// TIA Portal project "PID_TankLevel" (V16)

(* hardware
DEVICE "S71500/ET200MP-Station_1"  S7-1500 station
   slot 0: "Profilschiene_0"  6ES7 590-1***0-0AA0
   slot 1: "PLC_1"  CPU 1511-1 PN  6ES7 511-1AK00-0AB0  V1.8
   slot 2: "AI 8xU/I/RTD/TC ST_1"  AI 8xU/I/RTD/TC ST  6ES7 531-7KF00-0AB0  V2.0
   slot 3: "AI 8xU/I/RTD/TC ST_2"  AI 8xU/I/RTD/TC ST  6ES7 531-7KF00-0AB0  V2.0
   slot 4: "AI 8xU/I/RTD/TC ST_3"  AI 8xU/I/RTD/TC ST  6ES7 531-7KF00-0AB0  V2.0
   slot 5: "AI 8xU/I/RTD/TC ST_4"  AI 8xU/I/RTD/TC ST  6ES7 531-7KF00-0AB0  V2.0
   slot 6: "DI 16x24VDC BA_1"  DI 16x24VDC BA  6ES7 521-1BH10-0AA0  V1.0
*)

// ===== PLC "PLC_1"  CPU 1511-1 PN =====

VAR_GLOBAL   // PLC tag table "Standard-Variablentabelle"
   "System_Byte" AT %MB1 : Byte;
   "FirstScan" AT %M1.0 : Bool;
   "DiagStatusUpdate" AT %M1.1 : Bool;
   "AlwaysTRUE" AT %M1.2 : Bool;
   "AlwaysFALSE" AT %M1.3 : Bool;
   "Clock_Byte" AT %MB0 : Byte;
   "Clock_10Hz" AT %M0.0 : Bool;
   "Clock_5Hz" AT %M0.1 : Bool;
   "Clock_2.5Hz" AT %M0.2 : Bool;
   "Clock_2Hz" AT %M0.3 : Bool;
   "Clock_1.25Hz" AT %M0.4 : Bool;
   "Clock_1Hz" AT %M0.5 : Bool;
   "Clock_0.625Hz" AT %M0.6 : Bool;
   "Clock_0.5Hz" AT %M0.7 : Bool;
END_VAR

VAR_GLOBAL   // PLC tag table "INPUTS"
   "StartButton" AT %I0.0 : Bool;
   "ResetButton" AT %I0.1 : Bool;
   "StopButton" AT %I0.2 : Bool;
   "FactoryIORunning" AT %I0.3 : Bool;
   "LevelMeter" AT %ID30 : Real;
   "FlowMeter" AT %ID34 : Real;
   "SetPoint" AT %ID38 : Real;
END_VAR

VAR_GLOBAL   // PLC tag table "OUTPUTS"
   "StartLight" AT %Q0.0 : Bool;
   "ResetLight" AT %Q0.1 : Bool;
   "StopLight" AT %Q0.2 : Bool;
   "FillValve" AT %QD30 : Real;
   "DischargeValve" AT %QD34 : Real;
   "SP" AT %QD38 : DInt;
   "PV" AT %QD42 : DInt;
END_VAR

VAR_GLOBAL   // PLC tag table "SystemTags"
   "LevelMeter_Scaled" AT %MD30 : DInt;
   "FlowMeter_Scaled" AT %MD34 : DInt;
   "SetPoint_Scaled" AT %MD38 : DInt;
   "FillValve_Scaled" AT %MD42 : DInt;
   "DischargeValve_Scaled" AT %MD46 : DInt;
END_VAR

VAR_GLOBAL   // PLC tag table "GeneralTags"
   "System ON/OFF" AT %M100.0 : Bool;
END_VAR

ORGANIZATION_BLOCK "Main"   // OB1, LAD, ProgramCycle
TITLE = "Main Program Sweep (Cycle)"
{ S7_Optimized_Access := 'TRUE' }
VERSION : 0.1
   VAR_INPUT
      Initial_Call : Bool;   // Initial call of this OB
      Remanence : Bool;   // =True, if remanent data are available
   END_VAR
BEGIN

REGION Network 2
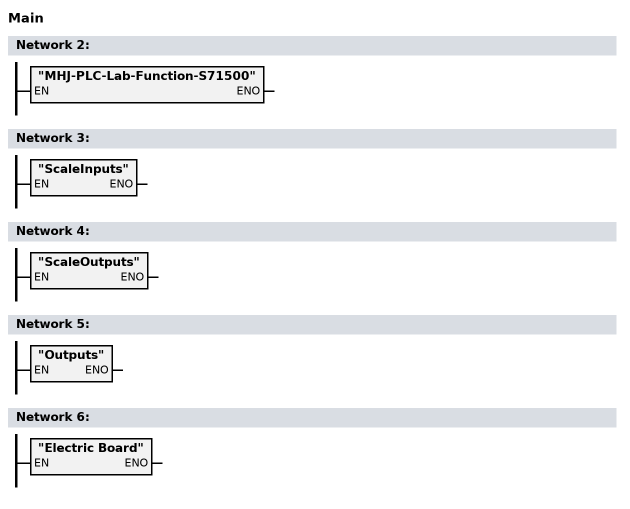
   RUNG wire#powerrail
      "MHJ-PLC-Lab-Function-S71500"()
   END_RUNG
   // the same network as SCL:
   "MHJ-PLC-Lab-Function-S71500"();
END_REGION

REGION Network 3
   RUNG wire#powerrail
      "ScaleInputs"()
   END_RUNG
   // the same network as SCL:
   "ScaleInputs"();
END_REGION

REGION Network 4
   RUNG wire#powerrail
      "ScaleOutputs"()
   END_RUNG
   // the same network as SCL:
   "ScaleOutputs"();
END_REGION

REGION Network 5
   RUNG wire#powerrail
      "Outputs"()
   END_RUNG
   // the same network as SCL:
   "Outputs"();
END_REGION

REGION Network 6
   RUNG wire#powerrail
      "Electric Board"()
   END_RUNG
   // the same network as SCL:
   "Electric Board"();
END_REGION
END_ORGANIZATION_BLOCK

// folder: INPUTS&OUTPUTS

FUNCTION "ScaleInputs" : Void   // FC1, LAD
{ S7_Optimized_Access := 'TRUE' }
VERSION : 0.1
   VAR_TEMP
      temp_levelmeter : Real;
      temp_setpoint : Real;
   END_VAR
BEGIN

REGION Network 2
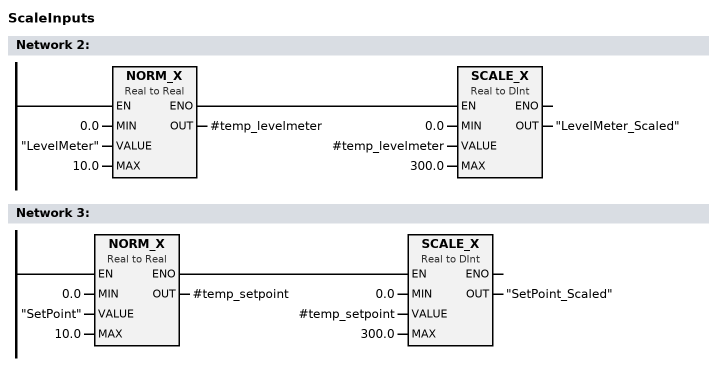
   RUNG wire#powerrail
      { S7_Templates := "[SrcType := Real, DestType := Real]" } Normalize(min := 0.0, value := "LevelMeter", max := 10.0, out => #temp_levelmeter)
      { S7_Templates := "[SrcType := Real, DestType := DInt]" } Scale(min := 0.0, value := #temp_levelmeter, max := 300.0, out => "LevelMeter_Scaled")
   END_RUNG
   // the same network as SCL:
   #temp_levelmeter := NORM_X(MIN := 0.0, VALUE := "LevelMeter", MAX := 10.0);
   "LevelMeter_Scaled" := SCALE_X(MIN := 0.0, VALUE := #temp_levelmeter, MAX := 300.0);
END_REGION

REGION Network 3
   RUNG wire#powerrail
      { S7_Templates := "[SrcType := Real, DestType := Real]" } Normalize(min := 0.0, value := "SetPoint", max := 10.0, out => #temp_setpoint)
      { S7_Templates := "[SrcType := Real, DestType := DInt]" } Scale(min := 0.0, value := #temp_setpoint, max := 300.0, out => "SetPoint_Scaled")
   END_RUNG
   // the same network as SCL:
   #temp_setpoint := NORM_X(MIN := 0.0, VALUE := "SetPoint", MAX := 10.0);
   "SetPoint_Scaled" := SCALE_X(MIN := 0.0, VALUE := #temp_setpoint, MAX := 300.0);
END_REGION
END_FUNCTION

FUNCTION "Outputs" : Void   // FC2, LAD
{ S7_Optimized_Access := 'TRUE' }
VERSION : 0.1
BEGIN

REGION Network 2
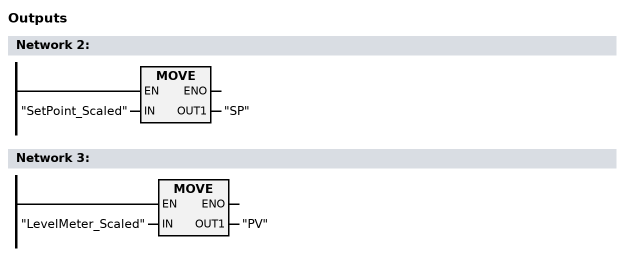
   RUNG wire#powerrail
      Move(in := "SetPoint_Scaled", out1 => "SP")
   END_RUNG
   // the same network as SCL:
   "SP" := "SetPoint_Scaled";
END_REGION

REGION Network 3
   RUNG wire#powerrail
      Move(in := "LevelMeter_Scaled", out1 => "PV")
   END_RUNG
   // the same network as SCL:
   "PV" := "LevelMeter_Scaled";
END_REGION
END_FUNCTION

FUNCTION "ScaleOutputs" : Void   // FC3, LAD
{ S7_Optimized_Access := 'TRUE' }
VERSION : 0.1
   VAR_TEMP
      temp_fillvalve : Real;
      temp_dischargevalve : Real;
   END_VAR
BEGIN

REGION Network 2
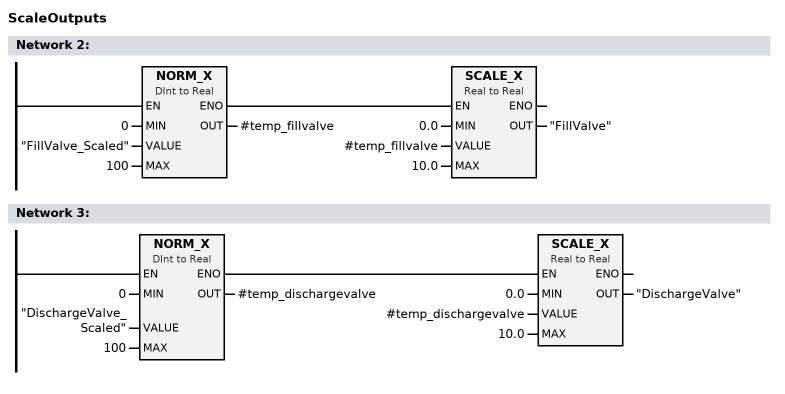
   RUNG wire#powerrail
      { S7_Templates := "[SrcType := DInt, DestType := Real]" } Normalize(min := 0, value := "FillValve_Scaled", max := 100, out => #temp_fillvalve)
      { S7_Templates := "[SrcType := Real, DestType := Real]" } Scale(min := 0.0, value := #temp_fillvalve, max := 10.0, out => "FillValve")
   END_RUNG
   // the same network as SCL:
   #temp_fillvalve := NORM_X(MIN := 0, VALUE := "FillValve_Scaled", MAX := 100);
   "FillValve" := SCALE_X(MIN := 0.0, VALUE := #temp_fillvalve, MAX := 10.0);
END_REGION

REGION Network 3
   RUNG wire#powerrail
      { S7_Templates := "[SrcType := DInt, DestType := Real]" } Normalize(min := 0, value := "DischargeValve_Scaled", max := 100, out => #temp_dischargevalve)
      { S7_Templates := "[SrcType := Real, DestType := Real]" } Scale(min := 0.0, value := #temp_dischargevalve, max := 10.0, out => "DischargeValve")
   END_RUNG
   // the same network as SCL:
   #temp_dischargevalve := NORM_X(MIN := 0, VALUE := "DischargeValve_Scaled", MAX := 100);
   "DischargeValve" := SCALE_X(MIN := 0.0, VALUE := #temp_dischargevalve, MAX := 10.0);
END_REGION
END_FUNCTION

// folder: SYSTEM BLOCKS

FUNCTION "Electric Board" : Void   // FC4, LAD
{ S7_Optimized_Access := 'TRUE' }
VERSION : 0.1
BEGIN

REGION Network 2
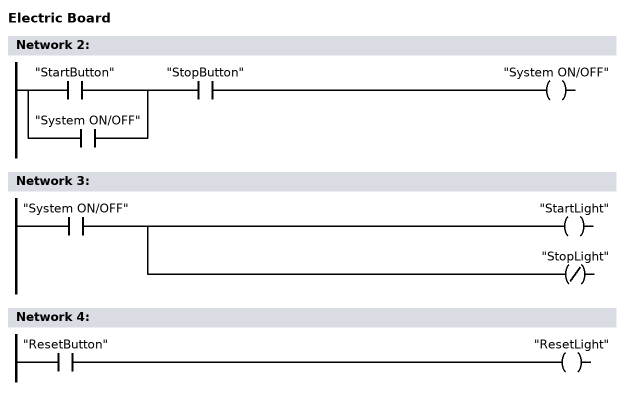
   RUNG wire#powerrail
      Contact( "StartButton" )
      wire#w1
      Contact( "StopButton" )
      Coil( "System ON/OFF" )
   END_RUNG
   RUNG wire#powerrail
      Contact( "System ON/OFF" )
   END_RUNG wire#w1
   // the same network as SCL:
   "System ON/OFF" := ("StartButton" OR "System ON/OFF") AND "StopButton";
END_REGION

REGION Network 3
   RUNG wire#powerrail
      Contact( "System ON/OFF" )
      wire#w1
      Coil( "StartLight" )
   END_RUNG
   RUNG wire#w1
      I_Coil( "StopLight" )
   END_RUNG
   // the same network as SCL:
   "StartLight" := "System ON/OFF";
   "StopLight" := NOT "System ON/OFF";
END_REGION

REGION Network 4
   RUNG wire#powerrail
      Contact( "ResetButton" )
      Coil( "ResetLight" )
   END_RUNG
   // the same network as SCL:
   "ResetLight" := "ResetButton";
END_REGION
END_FUNCTION

FUNCTION "MHJ-PLC-Lab-Function-S71500" : Void   // FC9000, SCL
{ S7_Optimized_Access := 'TRUE' }
VERSION : 0.1
   VAR_TEMP
      Value : Byte;
      ForCounter : Int;
   END_VAR
   VAR CONSTANT
      Value_01_DW : DWord := 16#1223_5486;
      Value_02_DW : DWord := 16#A6C9_D1F5;
   END_VAR
BEGIN

   #Value:=PEEK(area := 16#82,
        dbNumber := 0,
        byteOffset := 511);
   #Value := #Value + 1;

   POKE(area := 16#82,
        dbNumber := 0,
        byteOffset := 511,
        value := #Value);

   POKE(area := 16#82,
        dbNumber := 0,
        byteOffset := 1016,
        value := #Value_01_DW);
   POKE(area := 16#82,
        dbNumber := 0,
        byteOffset := 1020,
        value := #Value_02_DW);

   FOR #ForCounter := 0 TO 63 DO
       #Value:=PEEK(area := 16#1,
            dbNumber := 0,
            byteOffset := #ForCounter);
       POKE(area := 16#81,
            dbNumber := 0,
            byteOffset := #ForCounter,
            value := #Value);
   END_FOR;
   #Value := PEEK(area := 16#1,
                  dbNumber := 0,
                  byteOffset := 512);
   POKE(area := 16#82,
        dbNumber := 0,
        byteOffset := 512,
        value := #Value);
END_FUNCTION

ORGANIZATION_BLOCK "PID_LevelControl"   // OB30, LAD, CyclicInterrupt
{ S7_Optimized_Access := 'TRUE' }
VERSION : 0.1
   VAR_INPUT
      Initial_Call : Bool;   // Initial call of this OB
      Event_Count : Int;   // Events discarded
   END_VAR
   VAR_TEMP
      PID_Output : DInt;
      ABS_Output : DInt;
   END_VAR
BEGIN

REGION Network 2
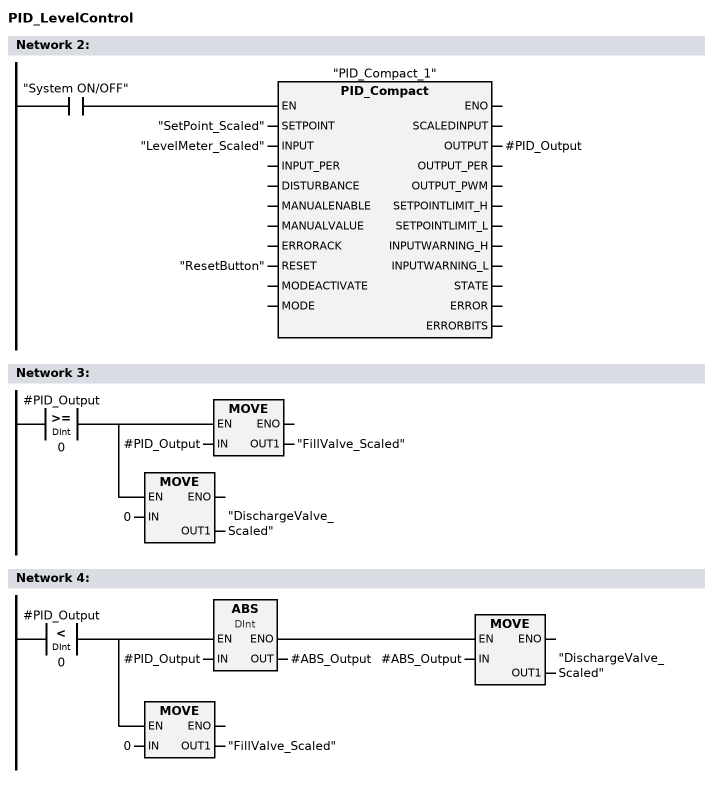
   IF "System ON/OFF" THEN
       "PID_Compact_1"(Setpoint := "SetPoint_Scaled",   // PID_Compact
                       Input := "LevelMeter_Scaled",
                       Reset := "ResetButton",
                       Output => #PID_Output);
   END_IF;
END_REGION

REGION Network 3
   RUNG wire#powerrail
      { S7_Templates := "SrcType := DInt" } GE_Contact(in1 := #PID_Output, in2 := 0)
      wire#w1
      Move(in := #PID_Output, out1 => "FillValve_Scaled")
   END_RUNG
   RUNG wire#w1
      Move(in := 0, out1 => "DischargeValve_Scaled")
   END_RUNG
   // the same network as SCL:
   IF #PID_Output >= 0 THEN
       "FillValve_Scaled" := #PID_Output;
       "DischargeValve_Scaled" := 0;
   END_IF;
END_REGION

REGION Network 4
   RUNG wire#powerrail
      { S7_Templates := "SrcType := DInt" } LT_Contact(in1 := #PID_Output, in2 := 0)
      wire#w1
      { S7_Templates := "SrcType := DInt" } Abs(in := #PID_Output, out => #ABS_Output)
      Move(in := #ABS_Output, out1 => "DischargeValve_Scaled")
   END_RUNG
   RUNG wire#w1
      Move(in := 0, out1 => "FillValve_Scaled")
   END_RUNG
   // the same network as SCL:
   IF #PID_Output < 0 THEN
       #ABS_Output := ABS(#PID_Output);
       "DischargeValve_Scaled" := #ABS_Output;
       "FillValve_Scaled" := 0;
   END_IF;
END_REGION
END_ORGANIZATION_BLOCK